FUNCTION_BLOCK fb_interface_bagmachine
VAR_INPUT
	bRun: BOOL;
	iPM	: INT;
	iBelt	: INT;
END_VAR
VAR_OUTPUT
END_VAR
VAR
END_VAR

IF bRun THEN
	GVL.pm[iPM].outConv.belt[iBelt].fbconverter.cmd	:= INT_TO_UINT(E_CMD_ConverterMotor.BACKWARE);
	GVL.pm[iPM].outConv.belt[iBelt].fbconverter.freq	:= 3500;	
ELSE
	GVL.pm[iPM].outConv.belt[iBelt].fbconverter.cmd	:= INT_TO_UINT(E_CMD_ConverterMotor.STOP);
	GVL.pm[iPM].outConv.belt[iBelt].fbconverter.freq	:= 0;
END_IF

END_FUNCTION_BLOCK

(* stored: Version 1.1.0.1, ProductVersion 3.1.4024.12
   POU fb_interface_bagmachine: Id {f060f8f2-ae65-4940-aac8-7b5b7fdaccc1}, SpecialFunc None *)
